// TIA Portal project "start-start" (V16)

(* hardware
DEVICE "S7-1200 station_1"  S7-1200 Station
   slot 0: "Rack_0"  S7-1200 Rack  Rack  V1.0
   slot 1: "PLC_1"  CPU 1212C AC/DC/Rly  6ES7 212-1BE40-0XB0  V4.0
*)

// ===== PLC "PLC_1"  CPU 1212C AC/DC/Rly =====

VAR_GLOBAL   // PLC tag table "Default tag table"
   "start" AT %I0.1 : Bool;
   "motor 1" AT %Q0.0 : Bool;
   "Tag_3" AT %M0.0 : Bool;
   "motor 2" AT %Q0.1 : Bool;
   "Tag_5" AT %M0.1 : Bool;
   "stop" AT %I0.0 : Bool;
   "Tag_1" AT %M0.2 : Bool;
END_VAR

ORGANIZATION_BLOCK "Main"   // OB1, LAD, ProgramCycle
TITLE = "Main Program Sweep (Cycle)"
{ S7_Optimized_Access := 'TRUE' }
VERSION : 0.1
   VAR_INPUT
      Initial_Call : Bool;   // Initial call of this OB
      Remanence : Bool;   // =True, if remanent data are available
   END_VAR
   VAR_TEMP   // added for the SCL form of the ladder/FBD networks
      _w1 : Bool;
   END_VAR
BEGIN

REGION Network 1
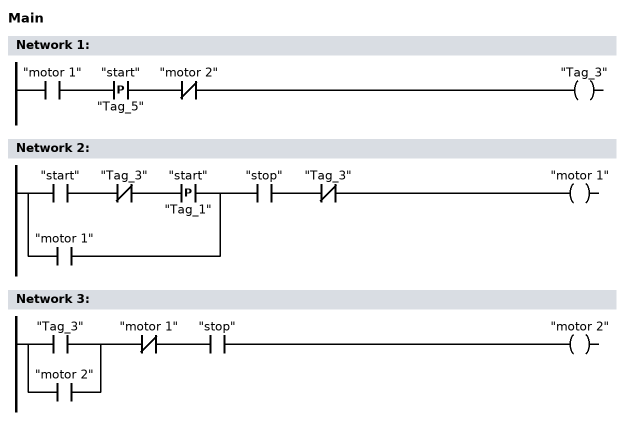
   RUNG wire#powerrail
      Contact( "motor 1" )
      P_Contact(operand := "start", bit := "Tag_5")
      I_Contact( "motor 2" )
      Coil( "Tag_3" )
   END_RUNG
   // the same network as SCL:
   #_w1 := "motor 1" AND "start" AND NOT "Tag_5";   // rising edge of "start"
   "Tag_5" := "start";
   "Tag_3" := #_w1 AND NOT "motor 2";
END_REGION

REGION Network 2
   RUNG wire#powerrail
      Contact( "start" )
      I_Contact( "Tag_3" )
      P_Contact(operand := "start", bit := "Tag_1")
      wire#w1
      Contact( "stop" )
      I_Contact( "Tag_3" )
      Coil( "motor 1" )
   END_RUNG
   RUNG wire#powerrail
      Contact( "motor 1" )
   END_RUNG wire#w1
   // the same network as SCL:
   #_w1 := "start" AND NOT "Tag_3" AND "start" AND NOT "Tag_1";   // rising edge of "start"
   "Tag_1" := "start";
   "motor 1" := (#_w1 OR "motor 1") AND "stop" AND NOT "Tag_3";
END_REGION

REGION Network 3
   RUNG wire#powerrail
      Contact( "Tag_3" )
      wire#w1
      I_Contact( "motor 1" )
      Contact( "stop" )
      Coil( "motor 2" )
   END_RUNG
   RUNG wire#powerrail
      Contact( "motor 2" )
   END_RUNG wire#w1
   // the same network as SCL:
   "motor 2" := ("Tag_3" OR "motor 2") AND NOT "motor 1" AND "stop";
END_REGION
END_ORGANIZATION_BLOCK